% RSLogix 500 project LGS3I_OVUN_CE_072417_WHAT_IS_THIS.RSS, saved by version 10.00.00.00 %
PROJECT "LVD4000"    % processor: MicroLogix 1400 %

PROGRAM FILES
  LAD 2 "MAIN"  45 rungs  % Main Program Routine %
  LAD 3 "BOT HSC"  3 rungs  % Bottom Conveyor High-Speed Counter Routine %
  LAD 4 "TOP HSC"  3 rungs  % Top Conveyor High-Speed Counter Routine %
  LAD 5 "BOT_TRACK"  2 rungs  % Bottom Conveyor Triggering & Tracking Sequence %
  LAD 6 "TOP_TRACK"  2 rungs  % Top Conveyor Triggering & Tracking Sequence %
  LAD 7 "STI_TRACK"  27 rungs
  LAD 8 "BOT_OPTIC"  5 rungs
  LAD 9 "SLOW_DATA"  12 rungs
  LAD 10 "BOT_NUT"  22 rungs
  LAD 11 "DATA_TRANS"  8 rungs
  LAD 12 "BOT_TRANSF"  2 rungs
  LAD 14 "TOP_OPTIC"  13 rungs
  LAD 16 "TOP_SIDE"  19 rungs
  LAD 20 "TOP_TOP"  30 rungs
  LAD 24 "TOP_BLOW"  6 rungs
  LAD 28 "FAULTS"  19 rungs
  LAD 29 "SPEED"  13 rungs
  LAD 30 "COUNT"  5 rungs
  LAD 31 "RATE"  1 rungs
  LAD 32 "LINEABOXER"  13 rungs
  LAD 33 "BULKBOXER"  3 rungs
  LAD 34 "CUSTBOXER"  12 rungs
  LAD 35 "CLEANUP"  9 rungs
  LAD 36 "J_CUST_BOX"  13 rungs  % Justin's customer boxing ladder %
  LAD 37 "BOXING"  12 rungs

DATA FILES
  O0 OUTPUT  11 elements
  I1 INPUT  11 elements
  S2 STATUS  66 elements
  B3 BINARY  15 elements
  T4 TIMER  40 elements
  C5 COUNTER  1 elements
  R6 CONTROL  10 elements
  N7 INTEGER  200 elements
  F8 FLOAT  100 elements
  B9 TOP BS DAT  256 elements
  B11 BOT BS DAT  256 elements
  L13  COUNTS  100 elements
  L23 NEW READ  100 elements
  L24 NEW WRITE  100 elements
  L42   52 elements

LADDER 2 "MAIN"    % Main Program Routine %
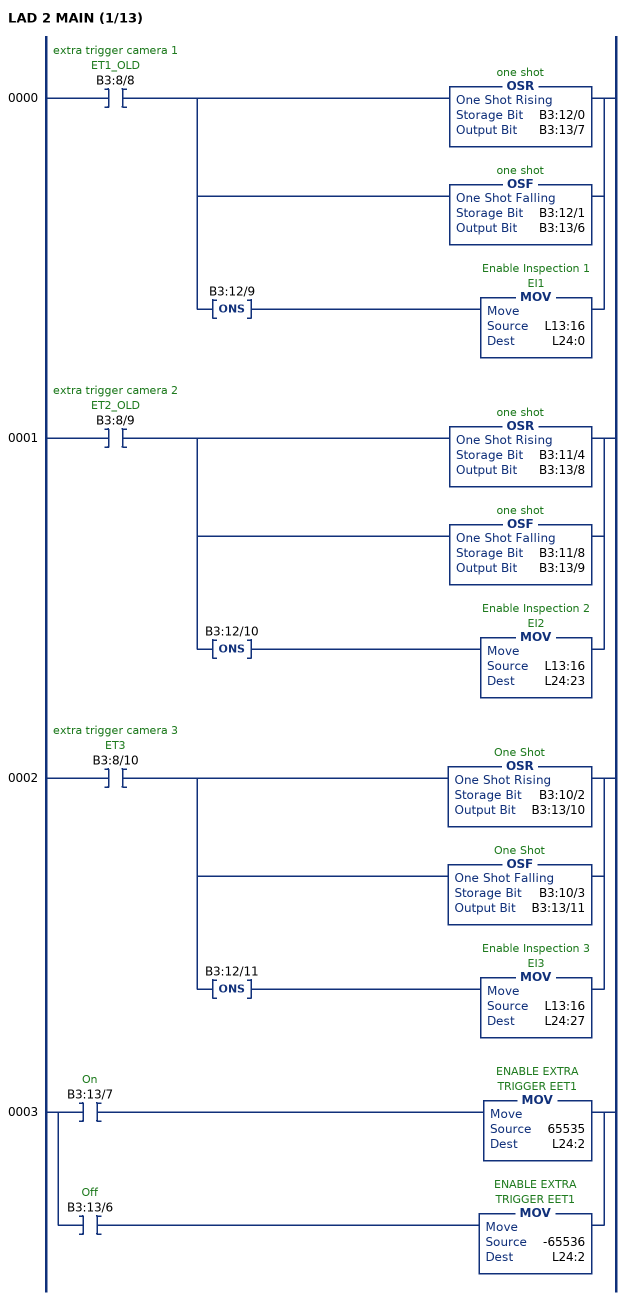
% Rung: 0 %
SOR XIC B3:8/8 BST OSR B3:12/0 B3:13/7 NXB OSF B3:12/1 B3:13/6 NXB ONS B3:12/9 MOV L13:16 L24:0 BND EOR
%   B3:8/8  ET1_OLD  "extra trigger camera 1" %
%   B3:12/0  "one shot" %
%   B3:13/7  "On" %
%   B3:12/1  "one shot" %
%   B3:13/6  "Off" %
%   L13:16  TRUE  "ONE TIME ENABLE FOR THE TIMES WHEN WE FORGET TO RE-ENABLE AFTER SHIPMENT" %
%   L24:0  EI1  "Enable Inspection 1" %
% Rung: 1 %
SOR XIC B3:8/9 BST OSR B3:11/4 B3:13/8 NXB OSF B3:11/8 B3:13/9 NXB ONS B3:12/10 MOV L13:16 L24:23 BND EOR
%   B3:8/9  ET2_OLD  "extra trigger camera 2" %
%   B3:11/4  "one shot" %
%   B3:13/8  "On" %
%   B3:11/8  "one shot" %
%   B3:13/9  "Off" %
%   L13:16  TRUE  "ONE TIME ENABLE FOR THE TIMES WHEN WE FORGET TO RE-ENABLE AFTER SHIPMENT" %
%   L24:23  EI2  "Enable Inspection 2" %
% Rung: 2 %
SOR XIC B3:8/10 BST OSR B3:10/2 B3:13/10 NXB OSF B3:10/3 B3:13/11 NXB ONS B3:12/11 MOV L13:16 L24:27 BND EOR
%   B3:8/10  ET3  "extra trigger camera 3" %
%   B3:10/2  "One Shot" %
%   B3:13/10  "On" %
%   B3:10/3  "One Shot" %
%   B3:13/11  "Off" %
%   L13:16  TRUE  "ONE TIME ENABLE FOR THE TIMES WHEN WE FORGET TO RE-ENABLE AFTER SHIPMENT" %
%   L24:27  EI3  "Enable Inspection 3" %
% Rung: 3 %
SOR BST XIC B3:13/7 MOV 65535 L24:2 NXB XIC B3:13/6 MOV -65536 L24:2 BND EOR
%   B3:13/7  "On" %
%   L24:2  EET1  "ENABLE EXTRA TRIGGER" %
%   B3:13/6  "Off" %

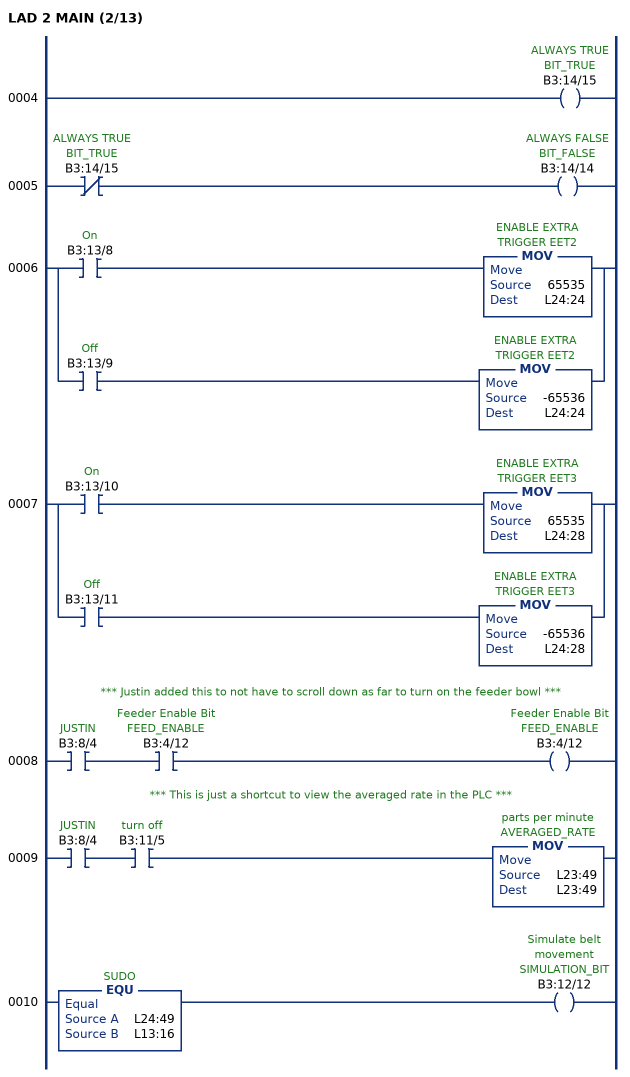
% Rung: 4 %
SOR OTE B3:14/15 EOR
%   B3:14/15  BIT_TRUE  "ALWAYS TRUE" %
% Rung: 5 %
SOR XIO B3:14/15 OTE B3:14/14 EOR
%   B3:14/15  BIT_TRUE  "ALWAYS TRUE" %
%   B3:14/14  BIT_FALSE  "ALWAYS FALSE" %
% Rung: 6 %
SOR BST XIC B3:13/8 MOV 65535 L24:24 NXB XIC B3:13/9 MOV -65536 L24:24 BND EOR
%   B3:13/8  "On" %
%   L24:24  EET2  "ENABLE EXTRA TRIGGER" %
%   B3:13/9  "Off" %
% Rung: 7 %
SOR BST XIC B3:13/10 MOV 65535 L24:28 NXB XIC B3:13/11 MOV -65536 L24:28 BND EOR
%   B3:13/10  "On" %
%   L24:28  EET3  "ENABLE EXTRA TRIGGER" %
%   B3:13/11  "Off" %
% Rung: 8 %
% *** Justin added this to not have to scroll down as far to turn on the feeder bowl *** %
SOR XIC B3:8/4 XIC B3:4/12 OTE B3:4/12 EOR
%   B3:8/4  JUSTIN %
%   B3:4/12  FEED_ENABLE  "Feeder Enable Bit" %
% Rung: 9 %
% *** This is just a shortcut to view the averaged rate in the PLC *** %
SOR XIC B3:8/4 XIC B3:11/5 MOV L23:49 L23:49 EOR
%   B3:8/4  JUSTIN %
%   B3:11/5  "turn off" %
%   L23:49  AVERAGED_RATE  "parts per minute" %
% Rung: 10 %
SOR EQU L24:49 L13:16 OTE B3:12/12 EOR
%   L24:49  SUDO %
%   L13:16  TRUE  "ONE TIME ENABLE FOR THE TIMES WHEN WE FORGET TO RE-ENABLE AFTER SHIPMENT" %
%   B3:12/12  SIMULATION_BIT  "Simulate belt movement" %

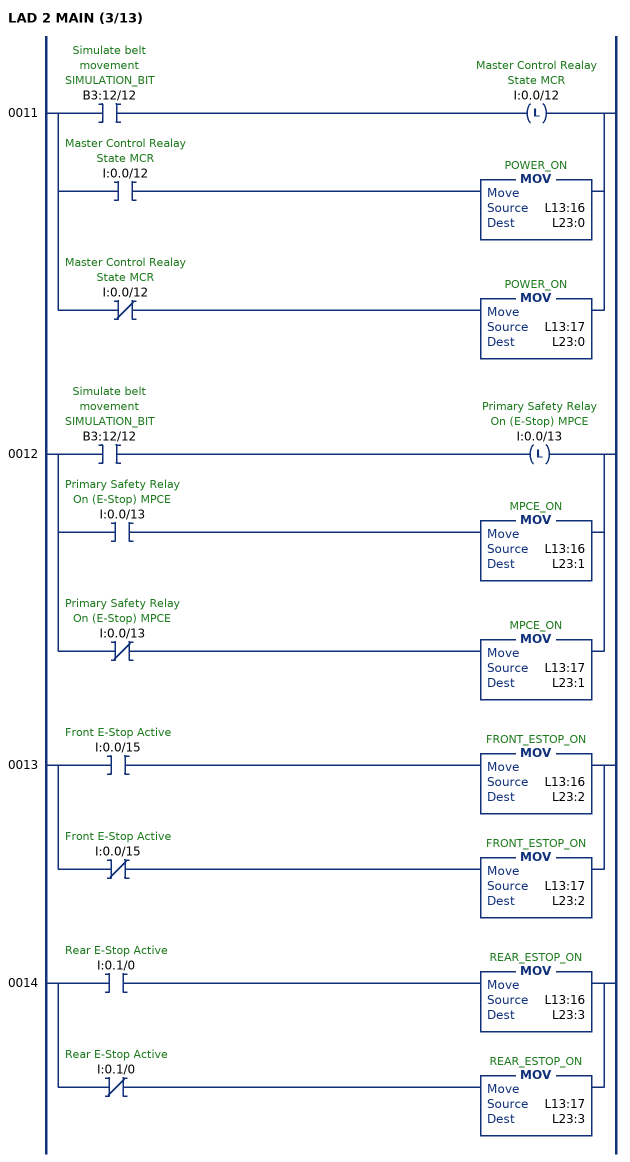
% Rung: 11 %
SOR BST XIC B3:12/12 OTL I:0.0/12 NXB XIC I:0.0/12 MOV L13:16 L23:0 NXB XIO I:0.0/12 MOV L13:17 L23:0 BND EOR
%   B3:12/12  SIMULATION_BIT  "Simulate belt movement" %
%   I:0.0/12  MCR  "Master Control Realay State" %
%   L13:16  TRUE  "ONE TIME ENABLE FOR THE TIMES WHEN WE FORGET TO RE-ENABLE AFTER SHIPMENT" %
%   L23:0  POWER_ON %
%   L13:17  FALSE %
% Rung: 12 %
SOR BST XIC B3:12/12 OTL I:0.0/13 NXB XIC I:0.0/13 MOV L13:16 L23:1 NXB XIO I:0.0/13 MOV L13:17 L23:1 BND EOR
%   B3:12/12  SIMULATION_BIT  "Simulate belt movement" %
%   I:0.0/13  MPCE  "Primary Safety Relay On (E-Stop)" %
%   L13:16  TRUE  "ONE TIME ENABLE FOR THE TIMES WHEN WE FORGET TO RE-ENABLE AFTER SHIPMENT" %
%   L23:1  MPCE_ON %
%   L13:17  FALSE %
% Rung: 13 %
SOR BST XIC I:0.0/15 MOV L13:16 L23:2 NXB XIO I:0.0/15 MOV L13:17 L23:2 BND EOR
%   I:0.0/15  "Front E-Stop Active" %
%   L13:16  TRUE  "ONE TIME ENABLE FOR THE TIMES WHEN WE FORGET TO RE-ENABLE AFTER SHIPMENT" %
%   L23:2  FRONT_ESTOP_ON %
%   L13:17  FALSE %
% Rung: 14 %
SOR BST XIC I:0.1/0 MOV L13:16 L23:3 NXB XIO I:0.1/0 MOV L13:17 L23:3 BND EOR
%   I:0.1/0  "Rear E-Stop Active" %
%   L13:16  TRUE  "ONE TIME ENABLE FOR THE TIMES WHEN WE FORGET TO RE-ENABLE AFTER SHIPMENT" %
%   L23:3  REAR_ESTOP_ON %
%   L13:17  FALSE %

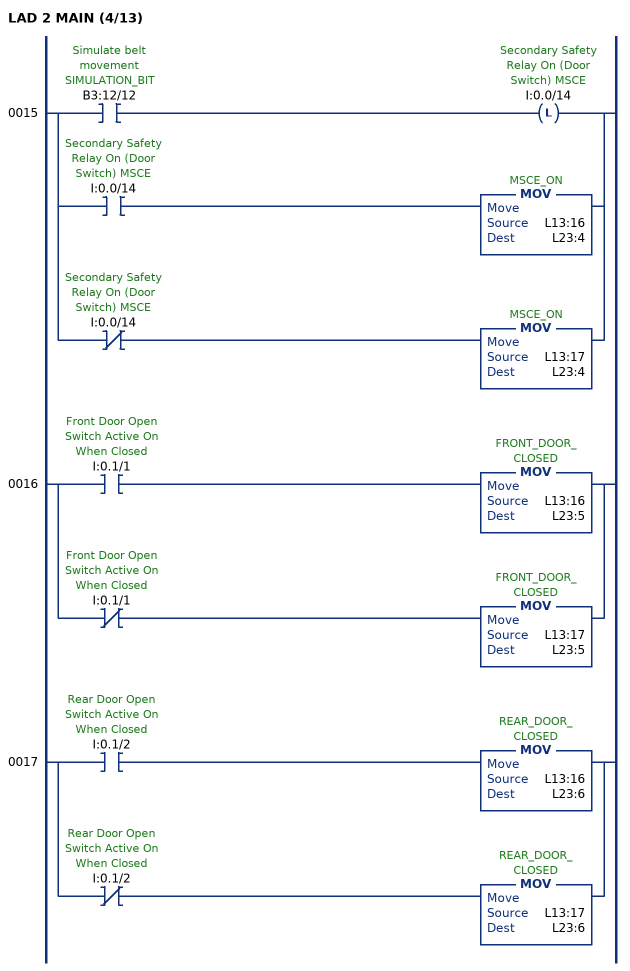
% Rung: 15 %
SOR BST XIC B3:12/12 OTL I:0.0/14 NXB XIC I:0.0/14 MOV L13:16 L23:4 NXB XIO I:0.0/14 MOV L13:17 L23:4 BND EOR
%   B3:12/12  SIMULATION_BIT  "Simulate belt movement" %
%   I:0.0/14  MSCE  "Secondary Safety Relay On (Door Switch)" %
%   L13:16  TRUE  "ONE TIME ENABLE FOR THE TIMES WHEN WE FORGET TO RE-ENABLE AFTER SHIPMENT" %
%   L23:4  MSCE_ON %
%   L13:17  FALSE %
% Rung: 16 %
SOR BST XIC I:0.1/1 MOV L13:16 L23:5 NXB XIO I:0.1/1 MOV L13:17 L23:5 BND EOR
%   I:0.1/1  "Front Door Open Switch Active On When Closed" %
%   L13:16  TRUE  "ONE TIME ENABLE FOR THE TIMES WHEN WE FORGET TO RE-ENABLE AFTER SHIPMENT" %
%   L23:5  FRONT_DOOR_CLOSED %
%   L13:17  FALSE %
% Rung: 17 %
SOR BST XIC I:0.1/2 MOV L13:16 L23:6 NXB XIO I:0.1/2 MOV L13:17 L23:6 BND EOR
%   I:0.1/2  "Rear Door Open Switch Active On When Closed" %
%   L13:16  TRUE  "ONE TIME ENABLE FOR THE TIMES WHEN WE FORGET TO RE-ENABLE AFTER SHIPMENT" %
%   L23:6  REAR_DOOR_CLOSED %
%   L13:17  FALSE %

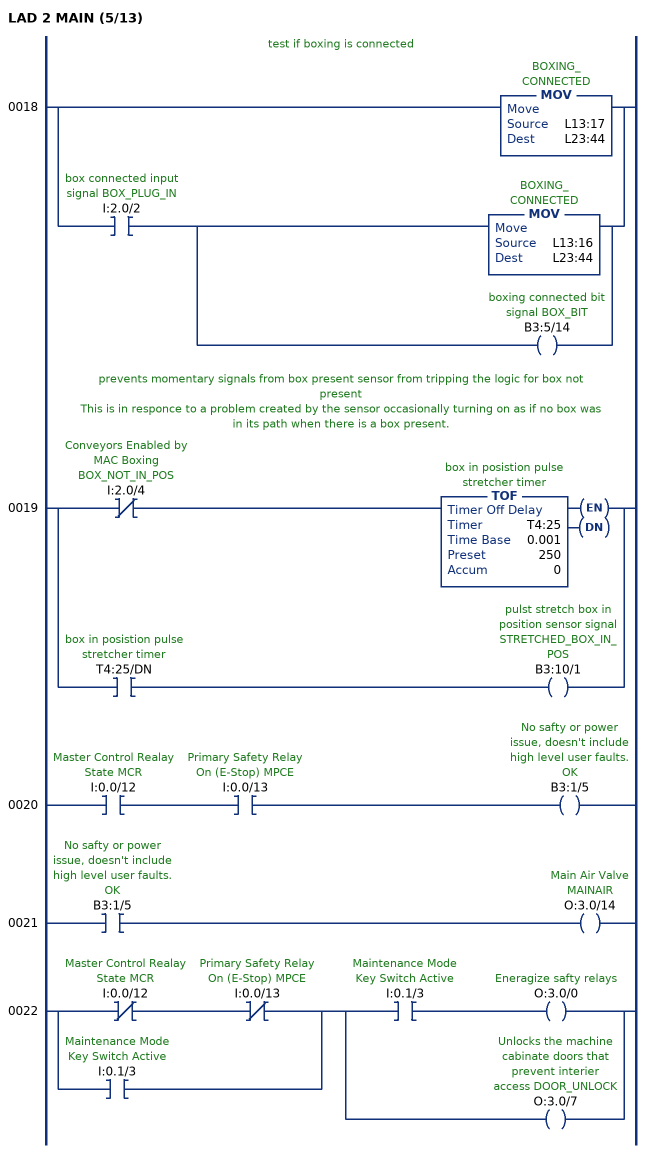
% Rung: 18 %
% test if boxing is connected %
SOR BST MOV L13:17 L23:44 NXB XIC I:2.0/2 BST MOV L13:16 L23:44 NXB OTE B3:5/14 BND BND EOR
%   L13:17  FALSE %
%   L23:44  BOXING_CONNECTED %
%   I:2.0/2  BOX_PLUG_IN  "box connected input signal" %
%   L13:16  TRUE  "ONE TIME ENABLE FOR THE TIMES WHEN WE FORGET TO RE-ENABLE AFTER SHIPMENT" %
%   B3:5/14  BOX_BIT  "boxing connected bit signal" %
% Rung: 19 %
% prevents momentary signals from box present sensor from tripping the logic for box not present
% 
% This is in responce to a problem created by the sensor occasionally turning on as if no box was in its path when there is a box present. %
SOR BST XIO I:2.0/4 TOF T4:25 0.001 250 0 NXB XIC T4:25/DN OTE B3:10/1 BND EOR
%   I:2.0/4  BOX_NOT_IN_POS  "Conveyors Enabled by MAC Boxing" %
%   T4:25  "box in posistion pulse stretcher timer" %
%   B3:10/1  STRETCHED_BOX_IN_POS  "pulst stretch box in position sensor signal" %
% Rung: 20 %
SOR XIC I:0.0/12 XIC I:0.0/13 OTE B3:1/5 EOR
%   I:0.0/12  MCR  "Master Control Realay State" %
%   I:0.0/13  MPCE  "Primary Safety Relay On (E-Stop)" %
%   B3:1/5  OK  "No safty or power issue, doesn't include high level user faults." %
% Rung: 21 %
SOR XIC B3:1/5 OTE O:3.0/14 EOR
%   B3:1/5  OK  "No safty or power issue, doesn't include high level user faults." %
%   O:3.0/14  MAINAIR  "Main Air Valve" %
% Rung: 22 %
SOR BST XIO I:0.0/12 XIO I:0.0/13 NXB XIC I:0.1/3 BND BST XIC I:0.1/3 OTE O:3.0/0 NXB OTE O:3.0/7 BND EOR
%   I:0.0/12  MCR  "Master Control Realay State" %
%   I:0.0/13  MPCE  "Primary Safety Relay On (E-Stop)" %
%   I:0.1/3  "Maintenance Mode Key Switch Active" %
%   O:3.0/0  "Eneragize safty relays" %
%   O:3.0/7  DOOR_UNLOCK  "Unlocks the machine cabinate doors that prevent interier access" %

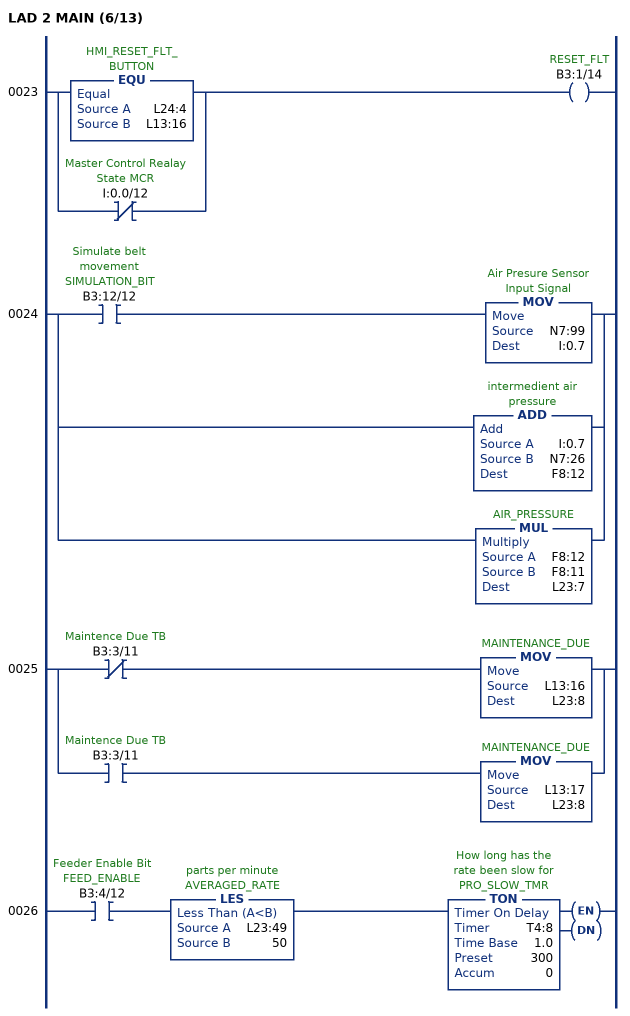
% Rung: 23 %
SOR BST EQU L24:4 L13:16 NXB XIO I:0.0/12 BND OTE B3:1/14 EOR
%   L24:4  HMI_RESET_FLT_BUTTON %
%   L13:16  TRUE  "ONE TIME ENABLE FOR THE TIMES WHEN WE FORGET TO RE-ENABLE AFTER SHIPMENT" %
%   I:0.0/12  MCR  "Master Control Realay State" %
%   B3:1/14  RESET_FLT %
% Rung: 24 %
SOR BST XIC B3:12/12 MOV N7:99 I:0.7 NXB ADD I:0.7 N7:26 F8:12 NXB MUL F8:12 F8:11 L23:7 BND EOR
%   B3:12/12  SIMULATION_BIT  "Simulate belt movement" %
%   I:0.7  "Air Presure Sensor Input Signal" %
%   N7:26  MAIN_AIR_OFFSET  "Main Air Offset old machine -398 new machine 0" %
%   F8:12  "intermedient air pressure" %
%   F8:11  AIR_MULTIPLIER  "main air multiplyer old machine 0.093" %
%   L23:7  AIR_PRESSURE %
% Rung: 25 %
SOR BST XIO B3:3/11 MOV L13:16 L23:8 NXB XIC B3:3/11 MOV L13:17 L23:8 BND EOR
%   B3:3/11  TB  "Maintence Due" %
%   L13:16  TRUE  "ONE TIME ENABLE FOR THE TIMES WHEN WE FORGET TO RE-ENABLE AFTER SHIPMENT" %
%   L23:8  MAINTENANCE_DUE %
%   L13:17  FALSE %
% Rung: 26 %
SOR XIC B3:4/12 LES L23:49 50 TON T4:8 1.0 300 0 EOR
%   B3:4/12  FEED_ENABLE  "Feeder Enable Bit" %
%   L23:49  AVERAGED_RATE  "parts per minute" %
%   T4:8  PRO_SLOW_TMR  "How long has the rate been slow for" %

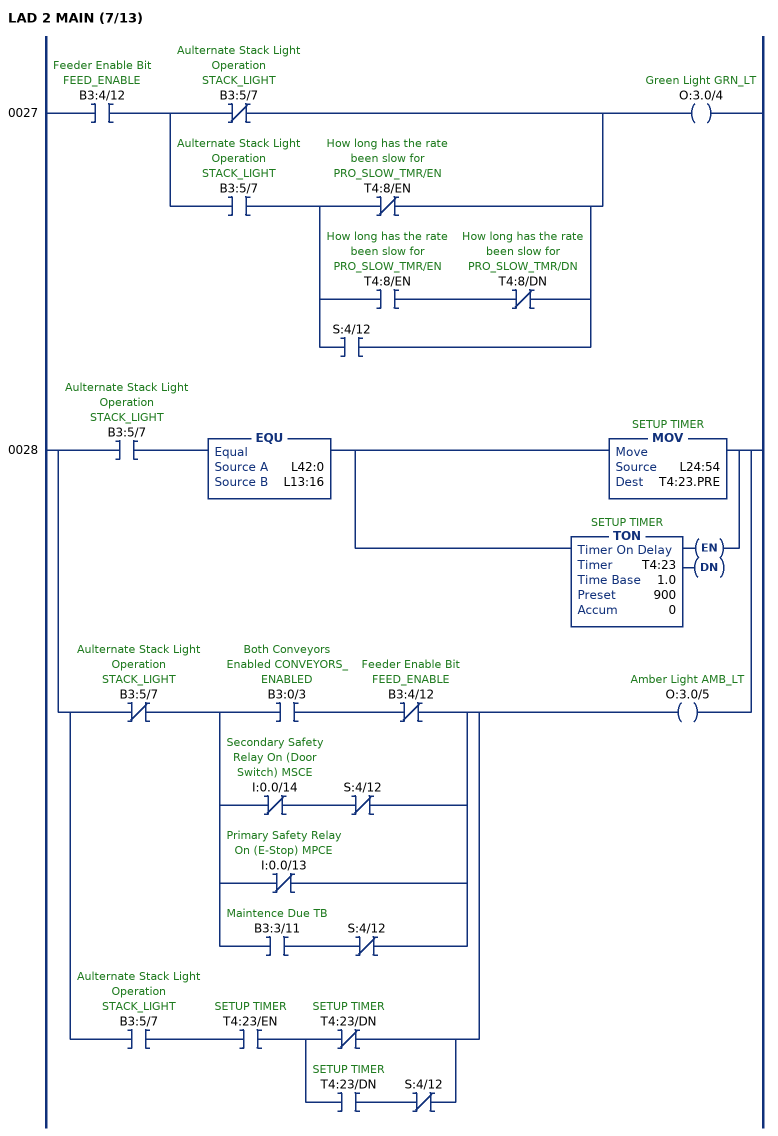
% Rung: 27 %
SOR XIC B3:4/12 BST XIO B3:5/7 NXB XIC B3:5/7 BST XIO T4:8/EN NXB XIC T4:8/EN XIO T4:8/DN NXB XIC S:4/12 BND BND OTE O:3.0/4 EOR
%   B3:4/12  FEED_ENABLE  "Feeder Enable Bit" %
%   B3:5/7  STACK_LIGHT  "Aulternate Stack Light Operation" %
%   T4:8  PRO_SLOW_TMR  "How long has the rate been slow for" %
%   O:3.0/4  GRN_LT  "Green Light" %
% Rung: 28 %
SOR BST XIC B3:5/7 EQU L42:0 L13:16 BST MOV L24:54 T4:23.PRE NXB TON T4:23 1.0 900 0 BND NXB BST XIO B3:5/7 BST XIC B3:0/3 XIO B3:4/12 NXB XIO I:0.0/14 XIO S:4/12 NXB XIO I:0.0/13 NXB XIC B3:3/11 XIO S:4/12 BND NXB XIC B3:5/7 XIC T4:23/EN BST XIO T4:23/DN NXB XIC T4:23/DN XIO S:4/12 BND BND OTE O:3.0/5 BND EOR
%   B3:5/7  STACK_LIGHT  "Aulternate Stack Light Operation" %
%   L13:16  TRUE  "ONE TIME ENABLE FOR THE TIMES WHEN WE FORGET TO RE-ENABLE AFTER SHIPMENT" %
%   L24:54  MAX_SETUP_TIME %
%   T4:23  "SETUP TIMER" %
%   B3:0/3  CONVEYORS_ENABLED  "Both Conveyors Enabled" %
%   B3:4/12  FEED_ENABLE  "Feeder Enable Bit" %
%   I:0.0/14  MSCE  "Secondary Safety Relay On (Door Switch)" %
%   I:0.0/13  MPCE  "Primary Safety Relay On (E-Stop)" %
%   B3:3/11  TB  "Maintence Due" %
%   O:3.0/5  AMB_LT  "Amber Light" %

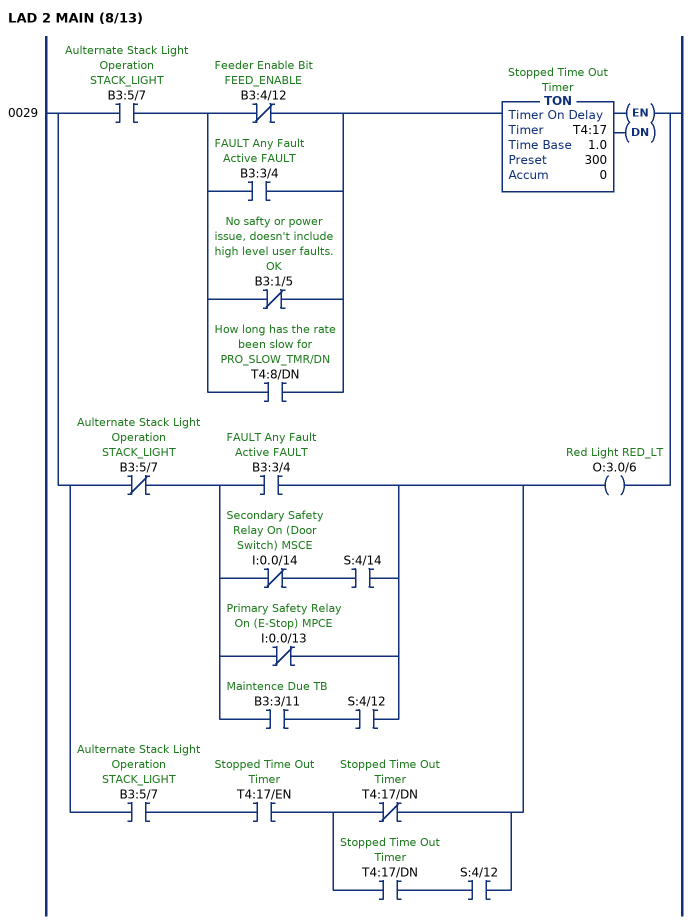
% Rung: 29 %
SOR BST XIC B3:5/7 BST XIO B3:4/12 NXB XIC B3:3/4 NXB XIO B3:1/5 NXB XIC T4:8/DN BND TON T4:17 1.0 300 0 NXB BST XIO B3:5/7 BST XIC B3:3/4 NXB XIO I:0.0/14 XIC S:4/14 NXB XIO I:0.0/13 NXB XIC B3:3/11 XIC S:4/12 BND NXB XIC B3:5/7 XIC T4:17/EN BST XIO T4:17/DN NXB XIC T4:17/DN XIC S:4/12 BND BND OTE O:3.0/6 BND EOR
%   B3:5/7  STACK_LIGHT  "Aulternate Stack Light Operation" %
%   B3:4/12  FEED_ENABLE  "Feeder Enable Bit" %
%   B3:3/4  FAULT  "FAULT Any Fault Active" %
%   B3:1/5  OK  "No safty or power issue, doesn't include high level user faults." %
%   T4:8  PRO_SLOW_TMR  "How long has the rate been slow for" %
%   T4:17  "Stopped Time Out Timer" %
%   I:0.0/14  MSCE  "Secondary Safety Relay On (Door Switch)" %
%   I:0.0/13  MPCE  "Primary Safety Relay On (E-Stop)" %
%   B3:3/11  TB  "Maintence Due" %
%   O:3.0/6  RED_LT  "Red Light" %

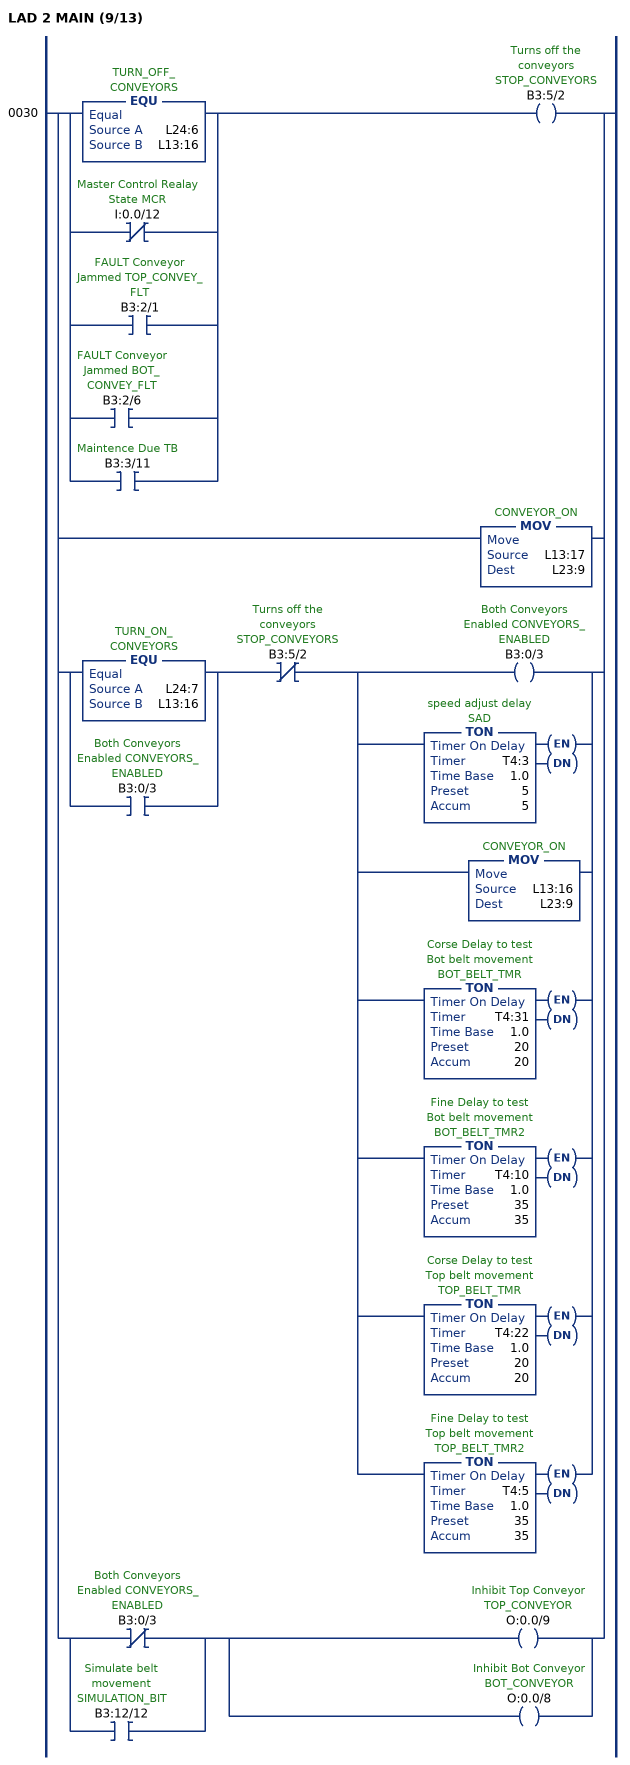
% Rung: 30 %
SOR BST BST EQU L24:6 L13:16 NXB XIO I:0.0/12 NXB XIC B3:2/1 NXB XIC B3:2/6 NXB XIC B3:3/11 BND OTE B3:5/2 NXB BST MOV L13:17 L23:9 NXB BST EQU L24:7 L13:16 NXB XIC B3:0/3 BND XIO B3:5/2 BST OTE B3:0/3 NXB TON T4:3 1.0 5 5 NXB MOV L13:16 L23:9 NXB TON T4:31 1.0 20 20 NXB TON T4:10 1.0 35 35 NXB TON T4:22 1.0 20 20 NXB TON T4:5 1.0 35 35 BND BND NXB BST XIO B3:0/3 NXB XIC B3:12/12 BND BST OTE O:0.0/9 NXB OTE O:0.0/8 BND BND EOR
%   L24:6  TURN_OFF_CONVEYORS %
%   L13:16  TRUE  "ONE TIME ENABLE FOR THE TIMES WHEN WE FORGET TO RE-ENABLE AFTER SHIPMENT" %
%   I:0.0/12  MCR  "Master Control Realay State" %
%   B3:2/1  "FAULT Conveyor Jammed TOP_CONVEY_FLT" %
%   B3:2/6  "FAULT Conveyor Jammed BOT_CONVEY_FLT" %
%   B3:3/11  TB  "Maintence Due" %
%   B3:5/2  STOP_CONVEYORS  "Turns off the conveyors" %
%   L13:17  FALSE %
%   L23:9  CONVEYOR_ON %
%   L24:7  TURN_ON_CONVEYORS %
%   B3:0/3  CONVEYORS_ENABLED  "Both Conveyors Enabled" %
%   T4:3  SAD  "speed adjust delay" %
%   T4:31  BOT_BELT_TMR  "Corse Delay to test Bot belt movement" %
%   T4:10  BOT_BELT_TMR2  "Fine Delay to test Bot belt movement" %
%   T4:22  TOP_BELT_TMR  "Corse Delay to test Top belt movement" %
%   T4:5  TOP_BELT_TMR2  "Fine Delay to test Top belt movement" %
%   B3:12/12  SIMULATION_BIT  "Simulate belt movement" %
%   O:0.0/9  TOP_CONVEYOR  "Inhibit Top Conveyor" %
%   O:0.0/8  BOT_CONVEYOR  "Inhibit Bot Conveyor" %

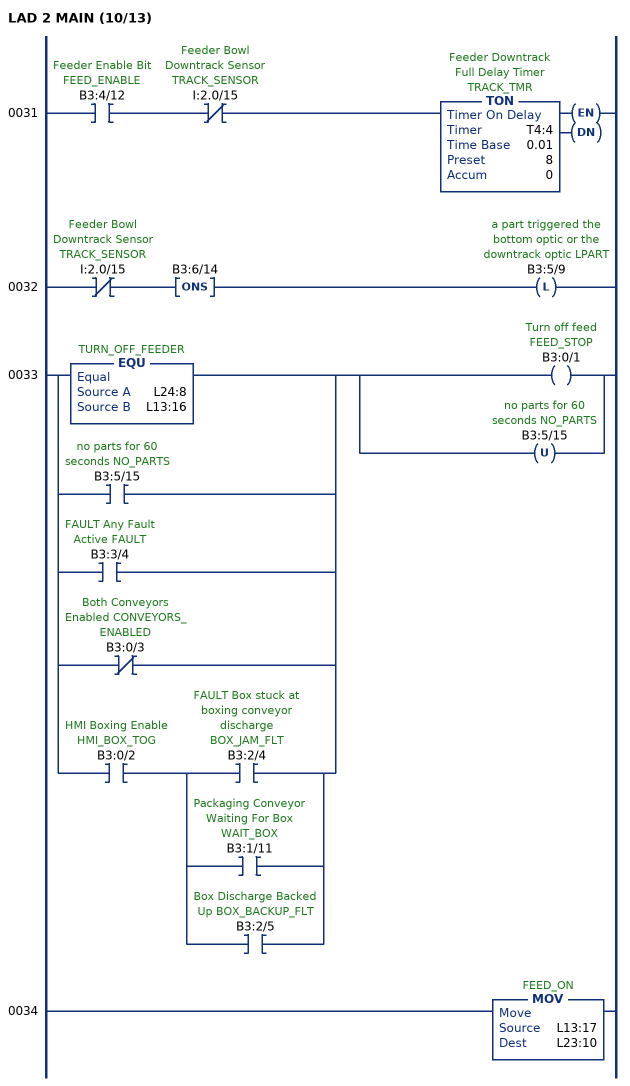
% Rung: 31 %
SOR XIC B3:4/12 XIO I:2.0/15 TON T4:4 0.01 8 0 EOR
%   B3:4/12  FEED_ENABLE  "Feeder Enable Bit" %
%   I:2.0/15  TRACK_SENSOR  "Feeder Bowl Downtrack Sensor" %
%   T4:4  TRACK_TMR  "Feeder Downtrack Full Delay Timer" %
% Rung: 32 %
SOR XIO I:2.0/15 ONS B3:6/14 OTL B3:5/9 EOR
%   I:2.0/15  TRACK_SENSOR  "Feeder Bowl Downtrack Sensor" %
%   B3:5/9  LPART  "a part triggered the bottom optic or the downtrack optic" %
% Rung: 33 %
SOR BST EQU L24:8 L13:16 NXB XIC B3:5/15 NXB XIC B3:3/4 NXB XIO B3:0/3 NXB XIC B3:0/2 BST XIC B3:2/4 NXB XIC B3:1/11 NXB XIC B3:2/5 BND BND BST OTE B3:0/1 NXB OTU B3:5/15 BND EOR
%   L24:8  TURN_OFF_FEEDER %
%   L13:16  TRUE  "ONE TIME ENABLE FOR THE TIMES WHEN WE FORGET TO RE-ENABLE AFTER SHIPMENT" %
%   B3:5/15  NO_PARTS  "no parts for 60 seconds" %
%   B3:3/4  FAULT  "FAULT Any Fault Active" %
%   B3:0/3  CONVEYORS_ENABLED  "Both Conveyors Enabled" %
%   B3:0/2  HMI_BOX_TOG  "HMI Boxing Enable" %
%   B3:2/4  BOX_JAM_FLT  "FAULT Box stuck at boxing conveyor discharge" %
%   B3:1/11  WAIT_BOX  "Packaging Conveyor Waiting For Box" %
%   B3:2/5  BOX_BACKUP_FLT  "Box Discharge Backed Up" %
%   B3:0/1  FEED_STOP  "Turn off feed" %
% Rung: 34 %
SOR MOV L13:17 L23:10 EOR
%   L13:17  FALSE %
%   L23:10  FEED_ON %

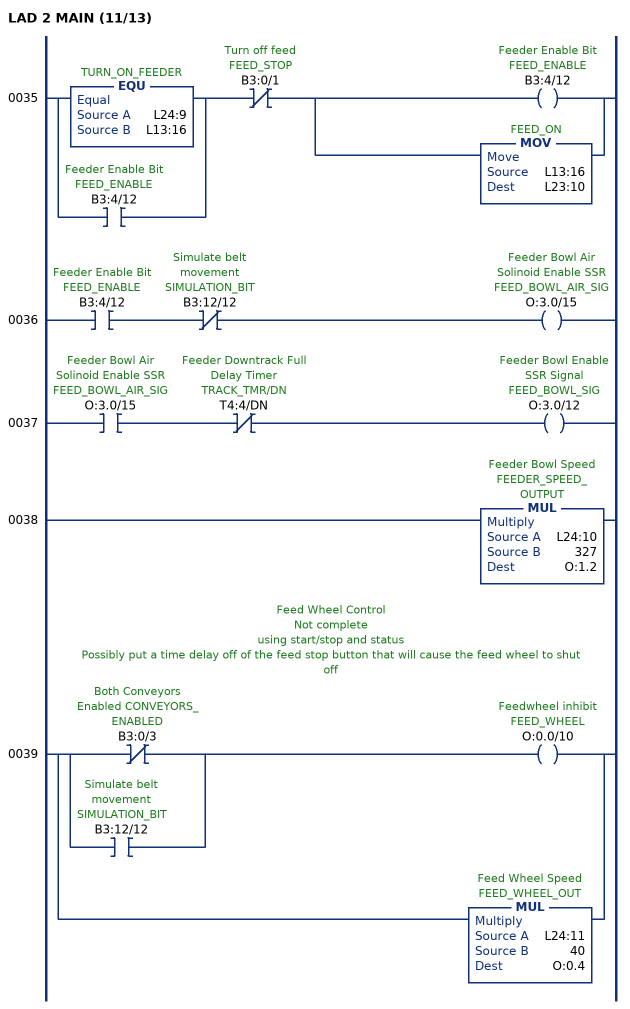
% Rung: 35 %
SOR BST EQU L24:9 L13:16 NXB XIC B3:4/12 BND XIO B3:0/1 BST OTE B3:4/12 NXB MOV L13:16 L23:10 BND EOR
%   L24:9  TURN_ON_FEEDER %
%   L13:16  TRUE  "ONE TIME ENABLE FOR THE TIMES WHEN WE FORGET TO RE-ENABLE AFTER SHIPMENT" %
%   B3:4/12  FEED_ENABLE  "Feeder Enable Bit" %
%   B3:0/1  FEED_STOP  "Turn off feed" %
%   L23:10  FEED_ON %
% Rung: 36 %
SOR XIC B3:4/12 XIO B3:12/12 OTE O:3.0/15 EOR
%   B3:4/12  FEED_ENABLE  "Feeder Enable Bit" %
%   B3:12/12  SIMULATION_BIT  "Simulate belt movement" %
%   O:3.0/15  FEED_BOWL_AIR_SIG  "Feeder Bowl Air Solinoid Enable SSR" %
% Rung: 37 %
SOR XIC O:3.0/15 XIO T4:4/DN OTE O:3.0/12 EOR
%   O:3.0/15  FEED_BOWL_AIR_SIG  "Feeder Bowl Air Solinoid Enable SSR" %
%   T4:4  TRACK_TMR  "Feeder Downtrack Full Delay Timer" %
%   O:3.0/12  FEED_BOWL_SIG  "Feeder Bowl Enable SSR Signal" %
% Rung: 38 %
SOR MUL L24:10 327 O:1.2 EOR
%   L24:10  FEEDER_SPEED %
%   O:1.2  FEEDER_SPEED_OUTPUT  "Feeder Bowl Speed" %
% Rung: 39 %
% Feed Wheel Control
% Not complete
% using start/stop and status
% Possibly put a time delay off of the feed stop button that will cause the feed wheel to shut off %
SOR BST BST XIO B3:0/3 NXB XIC B3:12/12 BND OTE O:0.0/10 NXB MUL L24:11 40 O:0.4 BND EOR
%   B3:0/3  CONVEYORS_ENABLED  "Both Conveyors Enabled" %
%   B3:12/12  SIMULATION_BIT  "Simulate belt movement" %
%   O:0.0/10  FEED_WHEEL  "Feedwheel inhibit" %
%   L24:11  FEED_WHEEL_SPEED %
%   O:0.4  FEED_WHEEL_OUT  "Feed Wheel Speed" %

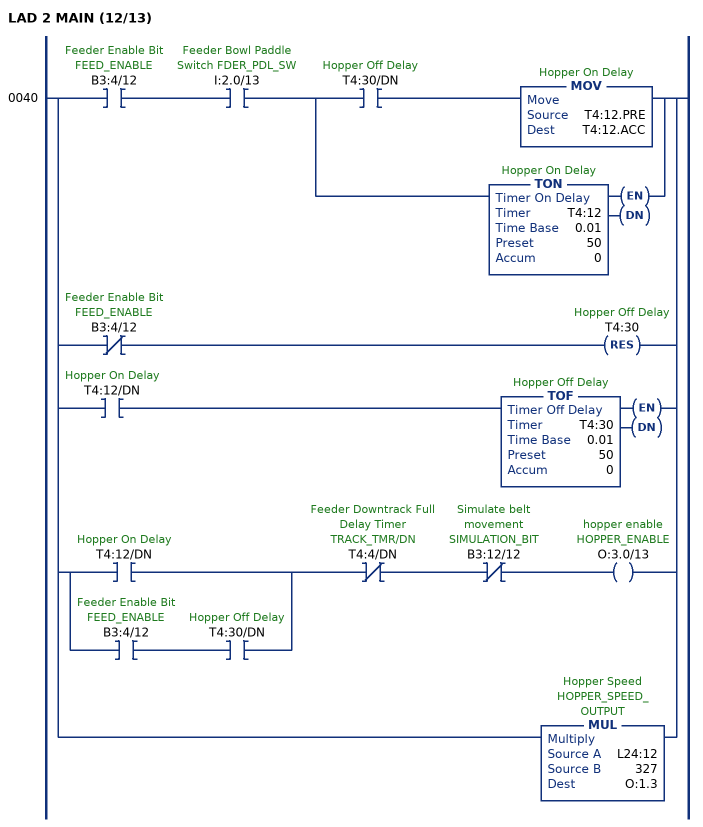
% Rung: 40 %
SOR BST XIC B3:4/12 XIC I:2.0/13 BST XIC T4:30/DN MOV T4:12.PRE T4:12.ACC NXB TON T4:12 0.01 50 0 BND NXB BST XIO B3:4/12 RES T4:30 NXB XIC T4:12/DN TOF T4:30 0.01 50 0 BND NXB BST XIC T4:12/DN NXB XIC B3:4/12 XIC T4:30/DN BND XIO T4:4/DN XIO B3:12/12 OTE O:3.0/13 NXB MUL L24:12 327 O:1.3 BND EOR
%   B3:4/12  FEED_ENABLE  "Feeder Enable Bit" %
%   I:2.0/13  FDER_PDL_SW  "Feeder Bowl Paddle Switch" %
%   T4:30  "Hopper Off Delay" %
%   T4:12  "Hopper On Delay" %
%   T4:4  TRACK_TMR  "Feeder Downtrack Full Delay Timer" %
%   B3:12/12  SIMULATION_BIT  "Simulate belt movement" %
%   O:3.0/13  HOPPER_ENABLE  "hopper enable" %
%   L24:12  HOPPER_SPEED %
%   O:1.3  HOPPER_SPEED_OUTPUT  "Hopper Speed" %

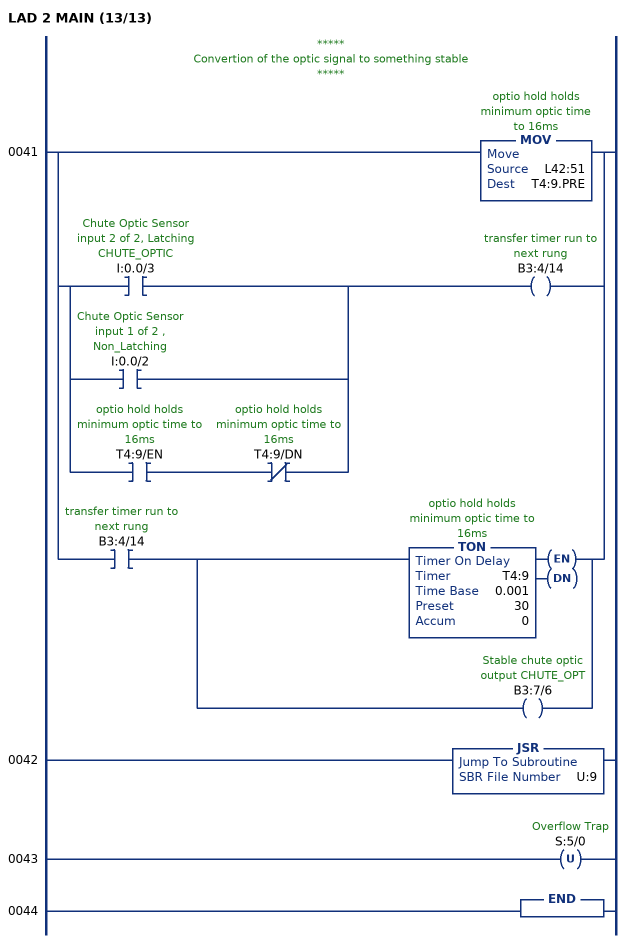
% Rung: 41 %
% *****
% Convertion of the optic signal to something stable
% ***** %
SOR BST MOV L42:51 T4:9.PRE NXB BST XIC I:0.0/3 NXB XIC I:0.0/2 NXB XIC T4:9/EN XIO T4:9/DN BND OTE B3:4/14 NXB XIC B3:4/14 BST TON T4:9 0.001 30 0 NXB OTE B3:7/6 BND BND EOR
%   L42:51  CHUTE_STABLIZING %
%   T4:9  "optio hold holds minimum optic time to 16ms" %
%   I:0.0/3  CHUTE_OPTIC  "Chute Optic Sensor input 2 of 2, Latching" %
%   I:0.0/2  "Chute Optic Sensor input 1 of 2 , Non_Latching" %
%   B3:4/14  "transfer timer run to next rung" %
%   B3:7/6  CHUTE_OPT  "Stable chute optic output" %
% Rung: 42 %
SOR JSR U:9 EOR
% Rung: 43 %
SOR OTU S:5/0 EOR
%   S:5/0  "Overflow Trap" %
% Rung: 44 %
SOR END EOR

LADDER 3 "BOT HSC"    % Bottom Conveyor High-Speed Counter Routine %
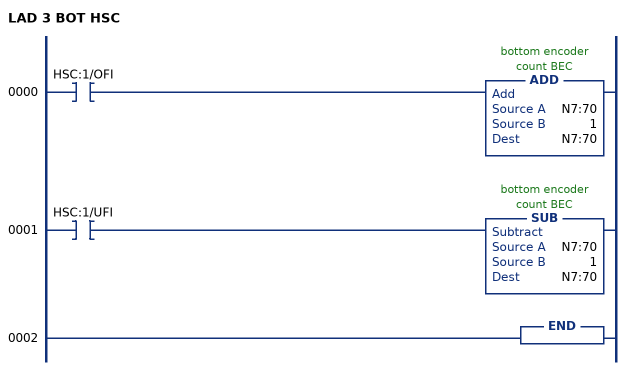
% Rung: 0 %
SOR XIC HSC:1/OFI ADD N7:70 1 N7:70 EOR
%   N7:70  BEC  "bottom encoder count" %
% Rung: 1 %
SOR XIC HSC:1/UFI SUB N7:70 1 N7:70 EOR
%   N7:70  BEC  "bottom encoder count" %
% Rung: 2 %
SOR END EOR

LADDER 4 "TOP HSC"    % Top Conveyor High-Speed Counter Routine %
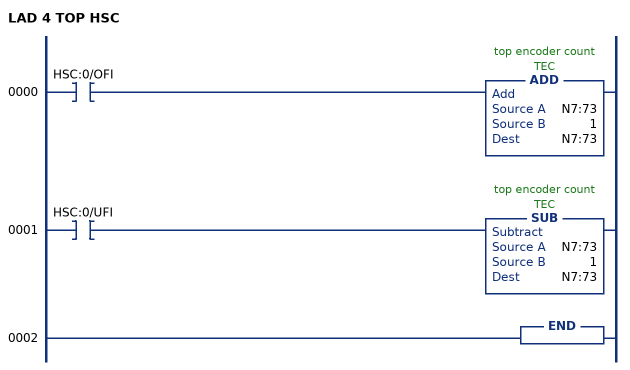
% Rung: 0 %
SOR XIC HSC:0/OFI ADD N7:73 1 N7:73 EOR
%   N7:73  TEC  "top encoder count" %
% Rung: 1 %
SOR XIC HSC:0/UFI SUB N7:73 1 N7:73 EOR
%   N7:73  TEC  "top encoder count" %
% Rung: 2 %
SOR END EOR

LADDER 5 "BOT_TRACK"    % Bottom Conveyor Triggering & Tracking Sequence %
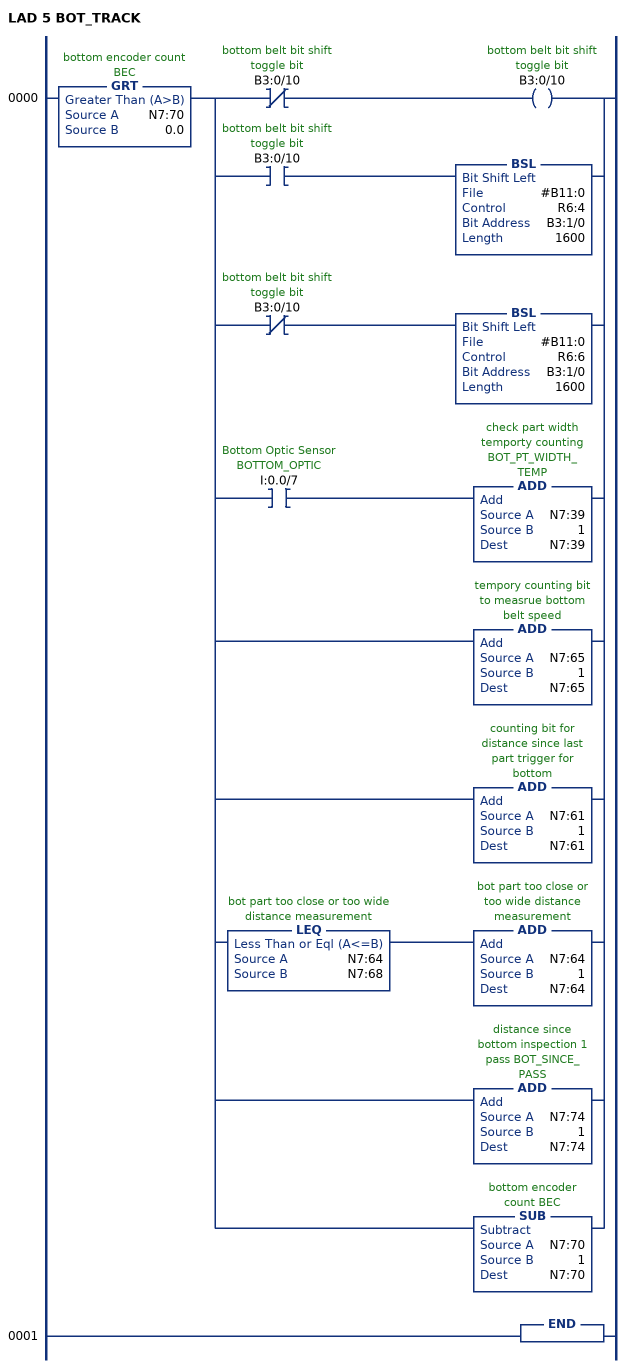
% Rung: 0 %
SOR GRT N7:70 0.0 BST XIO B3:0/10 OTE B3:0/10 NXB XIC B3:0/10 BSL #B11:0 R6:4 B3:1/0 1600 NXB XIO B3:0/10 BSL #B11:0 R6:6 B3:1/0 1600 NXB XIC I:0.0/7 ADD N7:39 1 N7:39 NXB ADD N7:65 1 N7:65 NXB ADD N7:61 1 N7:61 NXB LEQ N7:64 N7:68 ADD N7:64 1 N7:64 NXB ADD N7:74 1 N7:74 NXB SUB N7:70 1 N7:70 BND EOR
%   N7:70  BEC  "bottom encoder count" %
%   B3:0/10  "bottom belt bit shift toggle bit" %
%   B3:1/0  "Reserved For Shift Registers" %
%   I:0.0/7  BOTTOM_OPTIC  "Bottom Optic Sensor" %
%   N7:39  BOT_PT_WIDTH_TEMP  "check part width temporty counting" %
%   N7:65  "tempory counting bit to measrue bottom belt speed" %
%   N7:61  "counting bit for distance since last part trigger for bottom" %
%   N7:64  "bot part too close or too wide distance measurement" %
%   N7:68  "total distance to remove part present signals when parts are too close bottom" %
%   N7:74  BOT_SINCE_PASS  "distance since bottom inspection 1 pass" %
% Rung: 1 %
SOR END EOR

LADDER 6 "TOP_TRACK"    % Top Conveyor Triggering & Tracking Sequence %
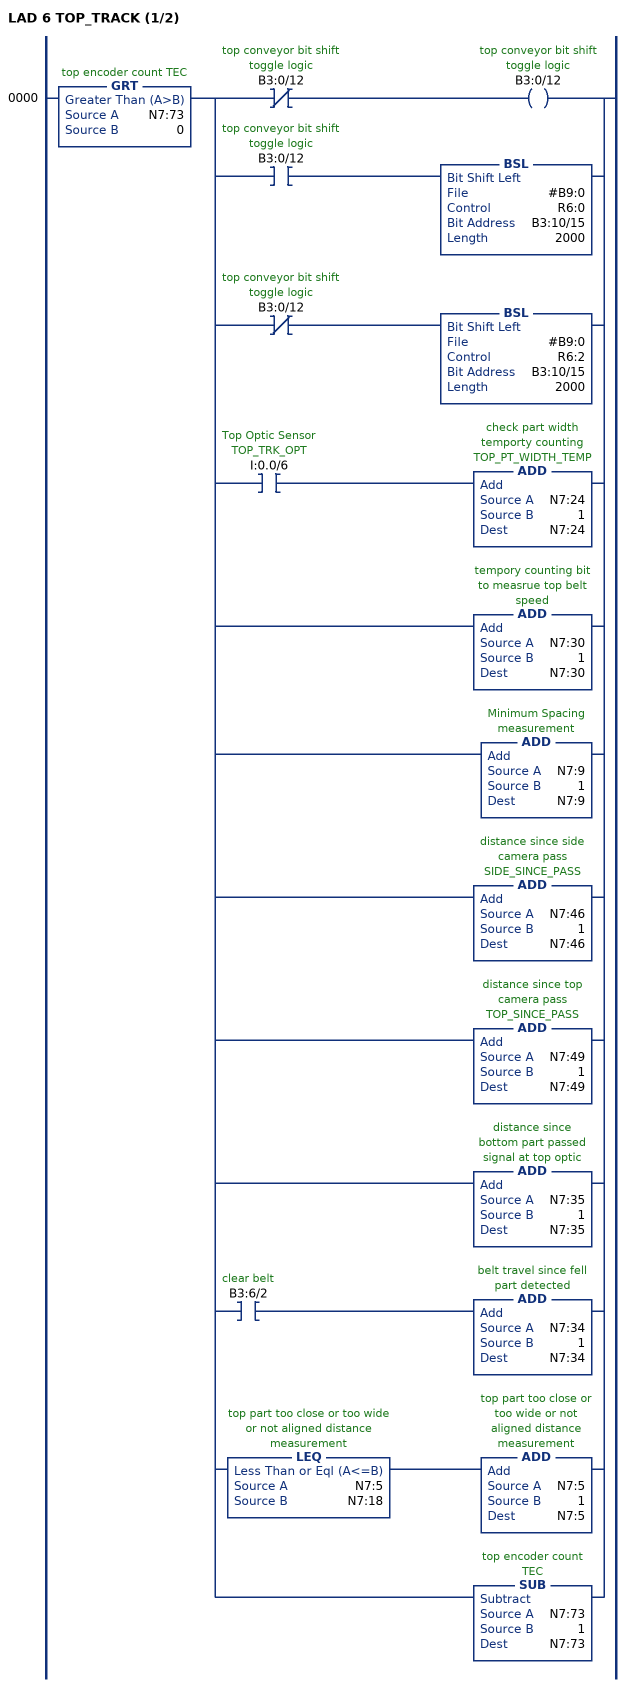
% Rung: 0 %
SOR GRT N7:73 0 BST XIO B3:0/12 OTE B3:0/12 NXB XIC B3:0/12 BSL #B9:0 R6:0 B3:10/15 2000 NXB XIO B3:0/12 BSL #B9:0 R6:2 B3:10/15 2000 NXB XIC I:0.0/6 ADD N7:24 1 N7:24 NXB ADD N7:30 1 N7:30 NXB ADD N7:9 1 N7:9 NXB ADD N7:46 1 N7:46 NXB ADD N7:49 1 N7:49 NXB ADD N7:35 1 N7:35 NXB XIC B3:6/2 ADD N7:34 1 N7:34 NXB LEQ N7:5 N7:18 ADD N7:5 1 N7:5 NXB SUB N7:73 1 N7:73 BND EOR
%   N7:73  TEC  "top encoder count" %
%   B3:0/12  "top conveyor bit shift toggle logic" %
%   R6:0  "Top Conveyor Part Tracking Bit Shit" %
%   B3:10/15  "Reserved For Shift Registers" %
%   I:0.0/6  TOP_TRK_OPT  "Top Optic Sensor" %
%   N7:24  TOP_PT_WIDTH_TEMP  "check part width temporty counting" %
%   N7:30  "tempory counting bit to measrue top belt speed" %
%   N7:9  "Minimum Spacing measurement" %
%   N7:46  SIDE_SINCE_PASS  "distance since side camera pass" %
%   N7:49  TOP_SINCE_PASS  "distance since top camera pass" %
%   N7:35  "distance since bottom part passed signal at top optic" %
%   B3:6/2  "clear belt" %
%   N7:34  "belt travel since fell part detected" %
%   N7:5  "top part too close or too wide or not aligned distance measurement" %
%   N7:18  "total distance to remove part present signals when parts are too close top" %

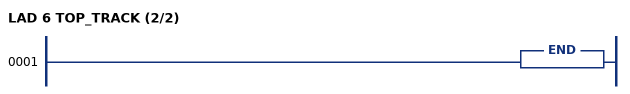
% Rung: 1 %
SOR END EOR

LADDER 7 "STI_TRACK"
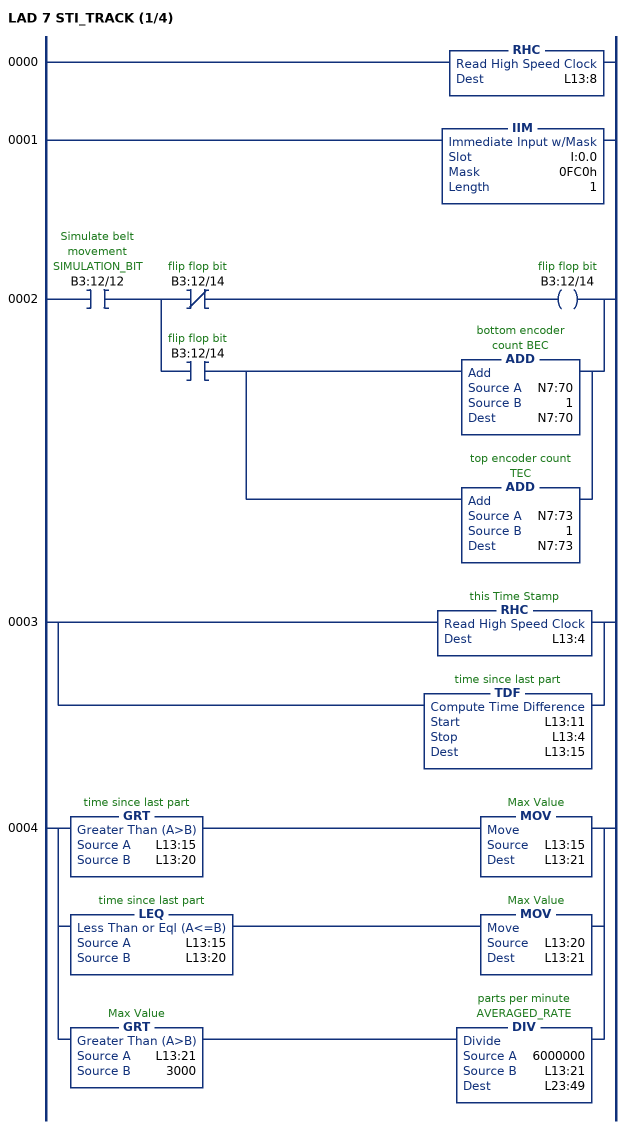
% Rung: 0 %
SOR RHC L13:8 EOR
% Rung: 1 %
SOR IIM I:0.0 0FC0h 1 EOR
% Rung: 2 %
SOR XIC B3:12/12 BST XIO B3:12/14 OTE B3:12/14 NXB XIC B3:12/14 BST ADD N7:70 1 N7:70 NXB ADD N7:73 1 N7:73 BND BND EOR
%   B3:12/12  SIMULATION_BIT  "Simulate belt movement" %
%   B3:12/14  "flip flop bit" %
%   N7:70  BEC  "bottom encoder count" %
%   N7:73  TEC  "top encoder count" %
% Rung: 3 %
SOR BST RHC L13:4 NXB TDF L13:11 L13:4 L13:15 BND EOR
%   L13:4  "this Time Stamp" %
%   L13:11  "Previous part time stamp" %
%   L13:15  "time since last part" %
% Rung: 4 %
SOR BST GRT L13:15 L13:20 MOV L13:15 L13:21 NXB LEQ L13:15 L13:20 MOV L13:20 L13:21 NXB GRT L13:21 3000 DIV 6000000 L13:21 L23:49 BND EOR
%   L13:15  "time since last part" %
%   L13:20  "last part to part time 10us" %
%   L13:21  "Max Value" %
%   L23:49  AVERAGED_RATE  "parts per minute" %

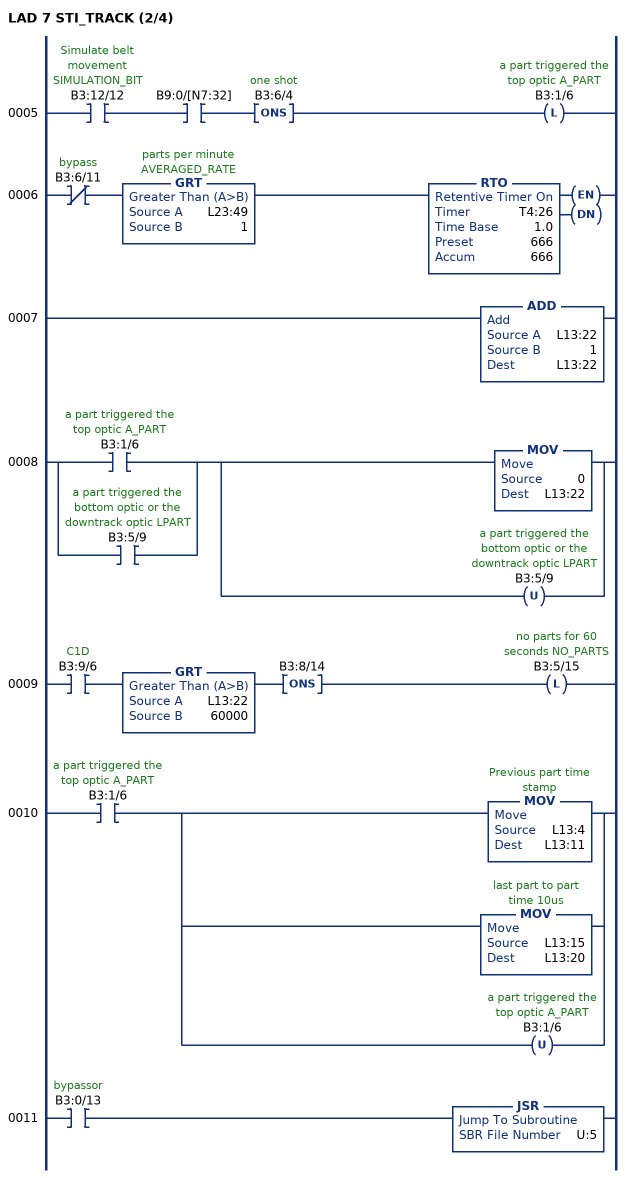
% Rung: 5 %
SOR XIC B3:12/12 XIC B9:0/[N7:32] ONS B3:6/4 OTL B3:1/6 EOR
%   B3:12/12  SIMULATION_BIT  "Simulate belt movement" %
%   N7:32  TOP_OPT_LOC  "Used As Indirect Address" %
%   B3:6/4  "one shot" %
%   B3:1/6  A_PART  "a part triggered the top optic" %
% Rung: 6 %
SOR XIO B3:6/11 GRT L23:49 1 RTO T4:26 1.0 666 666 EOR
%   B3:6/11  "bypass" %
%   L23:49  AVERAGED_RATE  "parts per minute" %
% Rung: 7 %
SOR ADD L13:22 1 L13:22 EOR
% Rung: 8 %
SOR BST XIC B3:1/6 NXB XIC B3:5/9 BND BST MOV 0 L13:22 NXB OTU B3:5/9 BND EOR
%   B3:1/6  A_PART  "a part triggered the top optic" %
%   B3:5/9  LPART  "a part triggered the bottom optic or the downtrack optic" %
% Rung: 9 %
SOR XIC B3:9/6 GRT L13:22 60000 ONS B3:8/14 OTL B3:5/15 EOR
%   B3:9/6  "C1D" %
%   B3:5/15  NO_PARTS  "no parts for 60 seconds" %
% Rung: 10 %
SOR XIC B3:1/6 BST MOV L13:4 L13:11 NXB MOV L13:15 L13:20 NXB OTU B3:1/6 BND EOR
%   B3:1/6  A_PART  "a part triggered the top optic" %
%   L13:4  "this Time Stamp" %
%   L13:11  "Previous part time stamp" %
%   L13:15  "time since last part" %
%   L13:20  "last part to part time 10us" %
% Rung: 11 %
SOR XIC B3:0/13 JSR U:5 EOR
%   B3:0/13  "bypassor" %

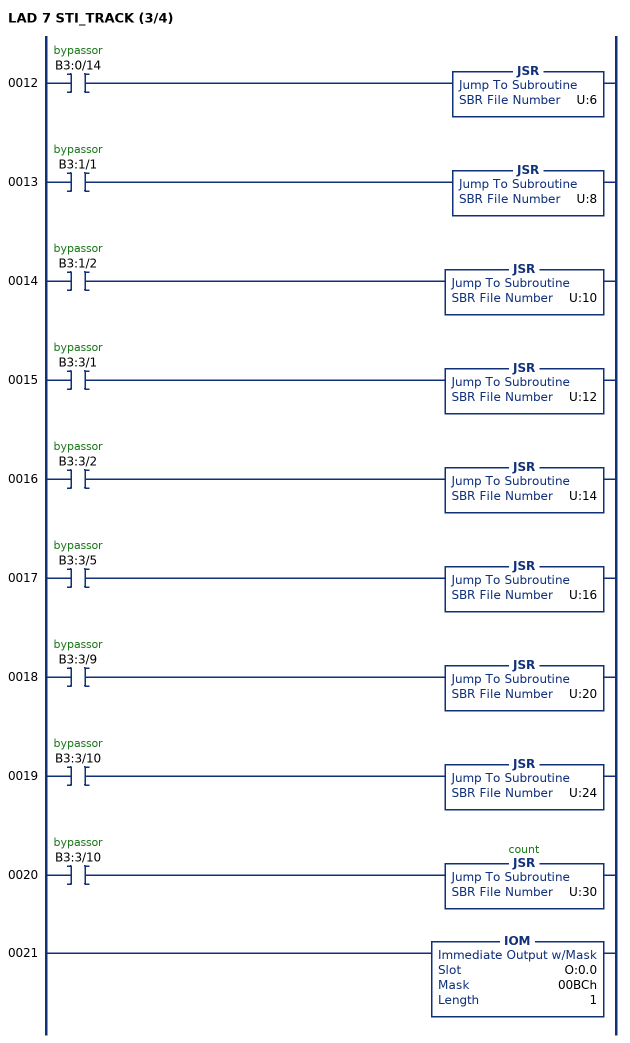
% Rung: 12 %
SOR XIC B3:0/14 JSR U:6 EOR
%   B3:0/14  "bypassor" %
% Rung: 13 %
SOR XIC B3:1/1 JSR U:8 EOR
%   B3:1/1  "bypassor" %
% Rung: 14 %
SOR XIC B3:1/2 JSR U:10 EOR
%   B3:1/2  "bypassor" %
% Rung: 15 %
SOR XIC B3:3/1 JSR U:12 EOR
%   B3:3/1  "bypassor" %
% Rung: 16 %
SOR XIC B3:3/2 JSR U:14 EOR
%   B3:3/2  "bypassor" %
% Rung: 17 %
SOR XIC B3:3/5 JSR U:16 EOR
%   B3:3/5  "bypassor" %
% Rung: 18 %
SOR XIC B3:3/9 JSR U:20 EOR
%   B3:3/9  "bypassor" %
% Rung: 19 %
SOR XIC B3:3/10 JSR U:24 EOR
%   B3:3/10  "bypassor" %
% Rung: 20 %
SOR XIC B3:3/10 JSR U:30 EOR
%   B3:3/10  "bypassor" %
%   U:30  "count" %
% Rung: 21 %
SOR IOM O:0.0 00BCh 1 EOR

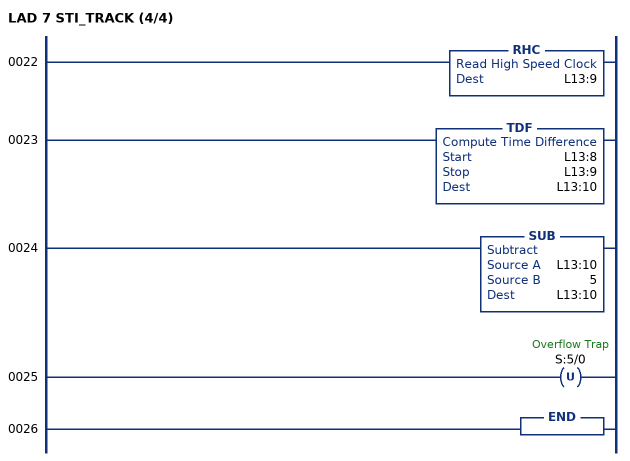
% Rung: 22 %
SOR RHC L13:9 EOR
% Rung: 23 %
SOR TDF L13:8 L13:9 L13:10 EOR
% Rung: 24 %
SOR SUB L13:10 5 L13:10 EOR
% Rung: 25 %
SOR OTU S:5/0 EOR
%   S:5/0  "Overflow Trap" %
% Rung: 26 %
SOR END EOR

LADDER 8 "BOT_OPTIC"
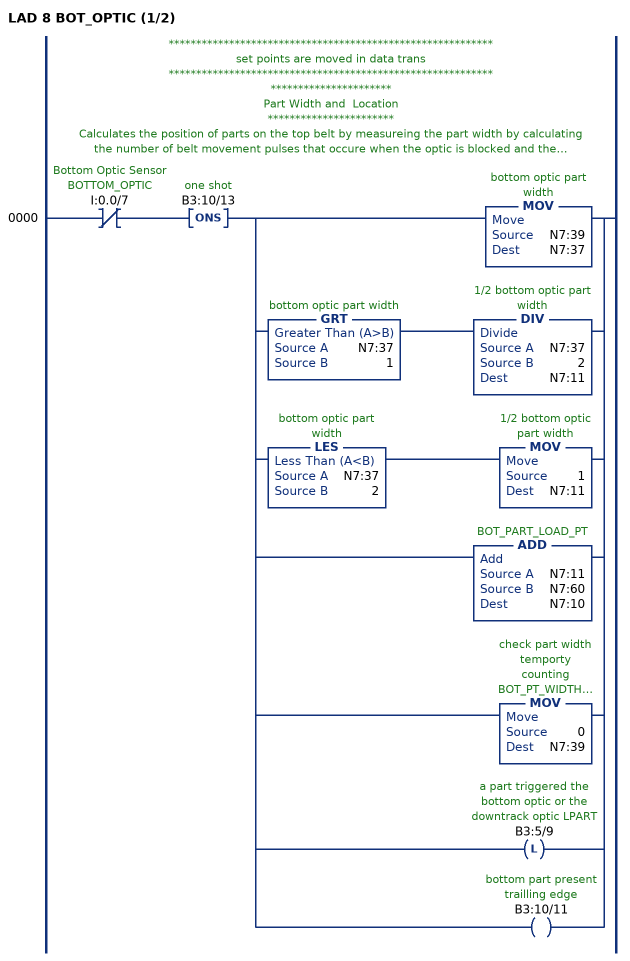
% Rung: 0 %
% ***********************************************************
% set points are moved in data trans
% ***********************************************************
% 
%  **********************
% Part Width and  Location
% ***********************
% 
% Calculates the position of parts on the top belt by measureing the part width by calculating the number of belt movement pulses that occure when the optic is blocked and then devides that in half and add that to the optic location in the part presnet bit shift when the top optic is cleared. %
SOR XIO I:0.0/7 ONS B3:10/13 BST MOV N7:39 N7:37 NXB GRT N7:37 1 DIV N7:37 2 N7:11 NXB LES N7:37 2 MOV 1 N7:11 NXB ADD N7:11 N7:60 N7:10 NXB MOV 0 N7:39 NXB OTL B3:5/9 NXB OTE B3:10/11 BND EOR
%   I:0.0/7  BOTTOM_OPTIC  "Bottom Optic Sensor" %
%   B3:10/13  "one shot" %
%   N7:39  BOT_PT_WIDTH_TEMP  "check part width temporty counting" %
%   N7:37  "bottom optic part width" %
%   N7:11  "1/2 bottom optic part width" %
%   N7:60  BOT_OPT_LOC  "bottom optic location" %
%   N7:10  BOT_PART_LOAD_PT %
%   B3:5/9  LPART  "a part triggered the bottom optic or the downtrack optic" %
%   B3:10/11  "bottom part present trailling edge" %

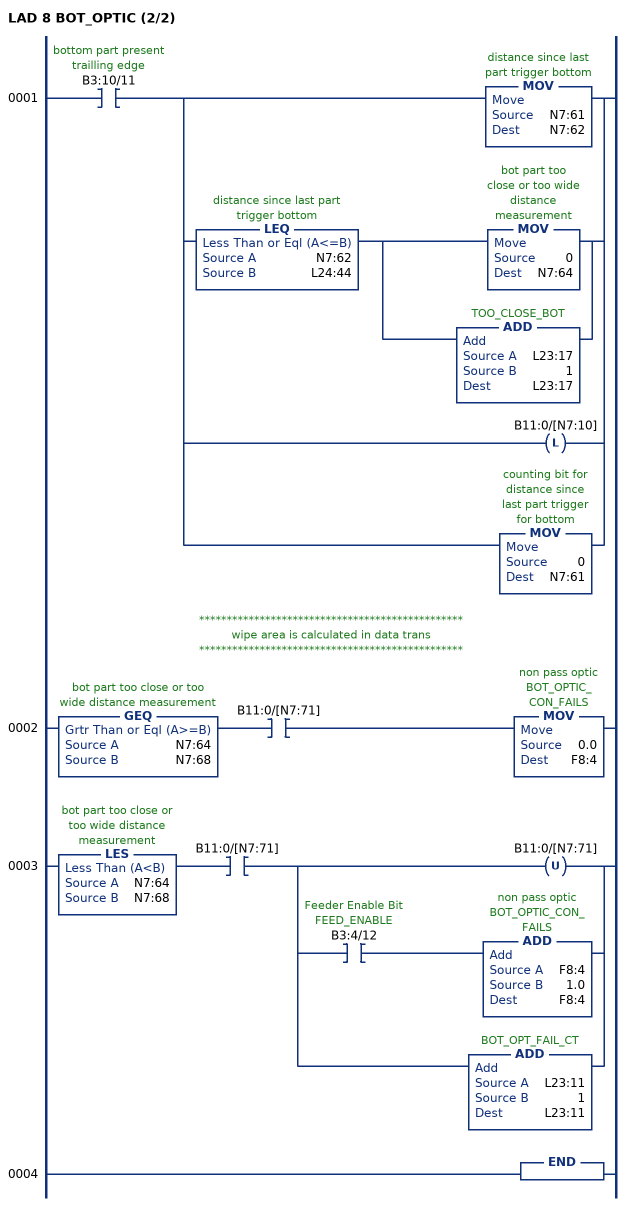
% Rung: 1 %
SOR XIC B3:10/11 BST MOV N7:61 N7:62 NXB LEQ N7:62 L24:44 BST MOV 0 N7:64 NXB ADD L23:17 1 L23:17 BND NXB OTL B11:0/[N7:10] NXB MOV 0 N7:61 BND EOR
%   B3:10/11  "bottom part present trailling edge" %
%   N7:61  "counting bit for distance since last part trigger for bottom" %
%   N7:62  "distance since last part trigger bottom" %
%   L24:44  MIN_PART_GAP_BOT %
%   N7:64  "bot part too close or too wide distance measurement" %
%   L23:17  TOO_CLOSE_BOT %
%   N7:10  BOT_PART_LOAD_PT %
% Rung: 2 %
% ************************************************
% wipe area is calculated in data trans
% ************************************************ %
SOR GEQ N7:64 N7:68 XIC B11:0/[N7:71] MOV 0.0 F8:4 EOR
%   N7:64  "bot part too close or too wide distance measurement" %
%   N7:68  "total distance to remove part present signals when parts are too close bottom" %
%   N7:71  BOT_PT_WIPE_LOC  "location to remove part present signals when signals are too close" %
%   F8:4  BOT_OPTIC_CON_FAILS  "non pass optic" %
% Rung: 3 %
SOR LES N7:64 N7:68 XIC B11:0/[N7:71] BST OTU B11:0/[N7:71] NXB XIC B3:4/12 ADD F8:4 1.0 F8:4 NXB ADD L23:11 1 L23:11 BND EOR
%   N7:64  "bot part too close or too wide distance measurement" %
%   N7:68  "total distance to remove part present signals when parts are too close bottom" %
%   N7:71  BOT_PT_WIPE_LOC  "location to remove part present signals when signals are too close" %
%   B3:4/12  FEED_ENABLE  "Feeder Enable Bit" %
%   F8:4  BOT_OPTIC_CON_FAILS  "non pass optic" %
%   L23:11  BOT_OPT_FAIL_CT %
% Rung: 4 %
SOR END EOR

LADDER 9 "SLOW_DATA"
